							IF aStatCommandQueue[nStatCommandIndex].nSubIndex = 0 THEN
								nStatOffset := 16;
							END_IF;
							nStatElement := 87;
							nStatBitLength := 16;
							bStatSource := False;
							JMP GetInteger;
						END_IF;
						// stProcessDataLimits - nUpper [UINT] [READ_ONLY]
						IF (aStatCommandQueue[nStatCommandIndex].nSubIndex = 0 AND nStatIndex = 1) OR (aStatCommandQueue[nStatCommandIndex].nSubIndex = 2 AND nStatIndex = 0) THEN
							IF aStatCommandQueue[nStatCommandIndex].nSubIndex = 0 THEN
								nStatOffset := 0;
							END_IF;
							nStatElement := 88;
							nStatBitLength := 16;
							bStatSource := False;
							JMP GetInteger;
						END_IF;
				// nSwitchCounter [UINT] [READ_ONLY]
					85:
						nStatComplex := cBASIC_TYPE;
						nStatBitLength := fbReadWriteReq.nCount;
						nStatElement := 89;
						JMP GetInteger;
				// nTemperatureInternal [INT] [READ_ONLY]
					86:
						nStatComplex := cBASIC_TYPE;
						nStatBitLength := fbReadWriteReq.nCount;
						nStatElement := 90;
						JMP GetInteger;
				// stNetwork [ComplexT] [READ_WRITE]
					88:
						nStatComplex := cCOMPLEX_RECORD_TYPE;
						nStatComplexDataTypeSize := UINT_TO_INT(aStatCommandQueue[nStatCommandIndex].nBitLength);
						nStatOffset := 0;
						// stNetwork - nRoleInNetwork [UINT] [READ_WRITE]
						IF (aStatCommandQueue[nStatCommandIndex].nSubIndex = 0 AND nStatIndex = 0) OR (aStatCommandQueue[nStatCommandIndex].nSubIndex = 1 AND nStatIndex = 0) THEN
							IF aStatCommandQueue[nStatCommandIndex].nSubIndex = 0 THEN
								nStatOffset := 8;
							END_IF;
							nStatElement := 91;
							nStatBitLength := 8;
							bStatSource := False;
							JMP GetInteger;
						END_IF;
						// stNetwork - nDeviceNoMasterHighestNo [UINT] [READ_WRITE]
						IF (aStatCommandQueue[nStatCommandIndex].nSubIndex = 0 AND nStatIndex = 1) OR (aStatCommandQueue[nStatCommandIndex].nSubIndex = 2 AND nStatIndex = 0) THEN
							IF aStatCommandQueue[nStatCommandIndex].nSubIndex = 0 THEN
								nStatOffset := 0;
							END_IF;
							nStatElement := 92;
							nStatBitLength := 8;
							bStatSource := False;
							JMP GetInteger;
						END_IF;
			END_CASE;
		END_IF;
		nStatState := cSTATE_JOB_FINISHED;
	END_IF;
// Update FB status
	IF nStatState = cSTATE_JOB_FINISHED THEN
		// Select next command
		nStatCommandIndex := nStatCommandIndex + 1;
		IF (nStatCommandIndex > cNUMBER_INPUTS) OR (aStatCommandQueue[nStatCommandIndex].nIndex = cEMPTY_COMMAND_QUEUE) THEN
			// Job done
			bDone := TRUE;
			bBusy := FALSE;
			bStatBusyMem := FALSE;
			bError := FALSE;
			stErrorCode.nAdsReadError := 16#0000;
			stErrorCode.nAdsWriteError := 16#0000;
			stErrorCode.nIndex := 0;
			stErrorCode.nSubIndex := 0;
			nStatState := cSTATE_READY;
			RETURN;
			// Next command
		ELSE
			nStatState := cSTATE_CLEAR_RECORD; // Send next IO-Link request
		END_IF;
	END_IF;
// End cycle
	RETURN;
// I/O mapping
	// SetInteger
		SetInteger:
			F_Leuze_IOL_SetInteger(nComplex := nStatComplex,
			                 nComplexDataTypeSize := nStatComplexDataTypeSize,
			                 nOffset := nStatOffset,
			                 nSource := nTempDeviceDataInteger,
			                 nBitLength := UINT_TO_INT(nStatBitLength),
			                 aIolRecords := aStatIOLRecords,
			                 aTempItems := aStatTempItems);
			IF (nStatComplex = cBASIC_TYPE) OR (nStatComplex = cCOMPLEX_RECORD_TYPE AND aStatCommandQueue[nStatCommandIndex].nSubIndex > 0) THEN
				fbReadWriteReq(bExecute := TRUE, bRW := TRUE, aData := aStatIOLRecords);
				nStatState := cSTATE_AWAIT_RESPONSE;
			ELSE
				nStatIndex := nStatIndex + 1;
			END_IF;
			RETURN;
	// SetBoolean
		SetBoolean:
			F_Leuze_IOL_SetBoolean(nComplex := nStatComplex,
			                     nComplexDataTypeSize := nStatComplexDataTypeSize,
			                     nOffset := nStatOffset,
			                     bSource := bTempDeviceDataBool,
			                     aIolRecords := aStatIOLRecords,
			                     aTempItems := aStatTempItems);
			IF (nStatComplex = cBASIC_TYPE) OR (nStatComplex = cCOMPLEX_RECORD_TYPE AND aStatCommandQueue[nStatCommandIndex].nSubIndex > 0) THEN
				fbReadWriteReq(bExecute := TRUE, bRW := TRUE, aData := aStatIOLRecords);
				nStatState := cSTATE_AWAIT_RESPONSE;
			ELSE
				nStatIndex := nStatIndex + 1;
			END_IF;
			RETURN;
	// SetString
		SetString:
			F_Leuze_IOL_SetString(nComplex := nStatComplex,
			                   nComplexDataTypeSize := nStatComplexDataTypeSize,
			                   nOffset := nStatOffset,
			                   nfixedLength := UINT_TO_INT(nStatBitLength),
			                   sSource := sTempDeviceDataString,
			                   aIolRecords := aStatIOLRecords,
			                   aTempItems := aStatTempItems);
			IF (nStatComplex = cBASIC_TYPE) OR (nStatComplex = cCOMPLEX_RECORD_TYPE AND aStatCommandQueue[nStatCommandIndex].nSubIndex > 0) THEN
				fbReadWriteReq(bExecute := TRUE, bRW := TRUE, aData := aStatIOLRecords);
				nStatState := cSTATE_AWAIT_RESPONSE;
			ELSE
				nStatIndex := nStatIndex + 1;
			END_IF;
			RETURN;
	// GetInteger
		GetInteger:
			nTempDeviceDataInteger := F_Leuze_IOL_GetInteger(nComplex := nStatComplex,
			                                               nComplexDataTypeSize := nStatComplexDataTypeSize,
			                                               nOffset := nStatOffset,
			                                               nBitLength := UINT_TO_INT(nStatBitLength),
			                                               bIsSigned := bStatSource,
			                                               aIolRecords := aStatIOLRecords,
			                                               aTempItems := aStatTempItems);
			IF nStatComplex = cCOMPLEX_ARRAY_TYPE THEN
				nStatOffset := nStatOffset + 1;
			END_IF;
			CASE nStatElement OF
				23:
						stDeviceData.stData.stDirectParametersPage1.nReserved_1 := DWORD_TO_UINT(nTempDeviceDataInteger);
				24:
						stDeviceData.stData.stDirectParametersPage1.nMasterCycleTime := DWORD_TO_UINT(nTempDeviceDataInteger);
				25:
						stDeviceData.stData.stDirectParametersPage1.nMinCycleTime := DWORD_TO_UINT(nTempDeviceDataInteger);
				26:
						stDeviceData.stData.stDirectParametersPage1.nMSequenceCapability := DWORD_TO_UINT(nTempDeviceDataInteger);
				27:
						stDeviceData.stData.stDirectParametersPage1.nIoLinkRevisionId := DWORD_TO_UINT(nTempDeviceDataInteger);
				28:
						stDeviceData.stData.stDirectParametersPage1.nProcessDataInputLength := DWORD_TO_UINT(nTempDeviceDataInteger);
				29:
						stDeviceData.stData.stDirectParametersPage1.nProcessDataOutputLength := DWORD_TO_UINT(nTempDeviceDataInteger);
				30:
						stDeviceData.stData.stDirectParametersPage1.nVendorId1 := DWORD_TO_UINT(nTempDeviceDataInteger);
				31:
						stDeviceData.stData.stDirectParametersPage1.nVendorId2 := DWORD_TO_UINT(nTempDeviceDataInteger);
				32:
						stDeviceData.stData.stDirectParametersPage1.nDeviceId1 := DWORD_TO_UINT(nTempDeviceDataInteger);
				33:
						stDeviceData.stData.stDirectParametersPage1.nDeviceId2 := DWORD_TO_UINT(nTempDeviceDataInteger);
				34:
						stDeviceData.stData.stDirectParametersPage1.nDeviceId3 := DWORD_TO_UINT(nTempDeviceDataInteger);
				35:
						stDeviceData.stData.stDirectParametersPage1.nReserved_13 := DWORD_TO_UINT(nTempDeviceDataInteger);
				36:
						stDeviceData.stData.stDirectParametersPage1.nReserved_14 := DWORD_TO_UINT(nTempDeviceDataInteger);
				37:
						stDeviceData.stData.stDirectParametersPage1.nReserved_15 := DWORD_TO_UINT(nTempDeviceDataInteger);
				39:
						stDeviceData.stData.stDirectParametersPage2.nDeviceSpecificParameter1 := DWORD_TO_UINT(nTempDeviceDataInteger);
				40:
						stDeviceData.stData.stDirectParametersPage2.nDeviceSpecificParameter2 := DWORD_TO_UINT(nTempDeviceDataInteger);
				41:
						stDeviceData.stData.stDirectParametersPage2.nDeviceSpecificParameter3 := DWORD_TO_UINT(nTempDeviceDataInteger);
				42:
						stDeviceData.stData.stDirectParametersPage2.nDeviceSpecificParameter4 := DWORD_TO_UINT(nTempDeviceDataInteger);
				43:
						stDeviceData.stData.stDirectParametersPage2.nDeviceSpecificParameter5 := DWORD_TO_UINT(nTempDeviceDataInteger);
				44:
						stDeviceData.stData.stDirectParametersPage2.nDeviceSpecificParameter6 := DWORD_TO_UINT(nTempDeviceDataInteger);
				45:
						stDeviceData.stData.stDirectParametersPage2.nDeviceSpecificParameter7 := DWORD_TO_UINT(nTempDeviceDataInteger);
				46:
						stDeviceData.stData.stDirectParametersPage2.nDeviceSpecificParameter8 := DWORD_TO_UINT(nTempDeviceDataInteger);
				47:
						stDeviceData.stData.stDirectParametersPage2.nDeviceSpecificParameter9 := DWORD_TO_UINT(nTempDeviceDataInteger);
				48:
						stDeviceData.stData.stDirectParametersPage2.nDeviceSpecificParameter10 := DWORD_TO_UINT(nTempDeviceDataInteger);
				49:
						stDeviceData.stData.stDirectParametersPage2.nDeviceSpecificParameter11 := DWORD_TO_UINT(nTempDeviceDataInteger);
				50:
						stDeviceData.stData.stDirectParametersPage2.nDeviceSpecificParameter12 := DWORD_TO_UINT(nTempDeviceDataInteger);
				51:
						stDeviceData.stData.stDirectParametersPage2.nDeviceSpecificParameter13 := DWORD_TO_UINT(nTempDeviceDataInteger);
				52:
						stDeviceData.stData.stDirectParametersPage2.nDeviceSpecificParameter14 := DWORD_TO_UINT(nTempDeviceDataInteger);
				53:
						stDeviceData.stData.stDirectParametersPage2.nDeviceSpecificParameter15 := DWORD_TO_UINT(nTempDeviceDataInteger);
				54:
						stDeviceData.stData.stDirectParametersPage2.nDeviceSpecificParameter16 := DWORD_TO_UINT(nTempDeviceDataInteger);
				67:
						stDeviceData.stData.nErrorCount := DWORD_TO_UINT(nTempDeviceDataInteger);
				68:
						stDeviceData.stData.nDeviceStatus := DWORD_TO_UINT(nTempDeviceDataInteger);
				69:
						stDeviceData.stData.stTeachState.nTeachState := DWORD_TO_UINT(nTempDeviceDataInteger);
				70:
						stDeviceData.stData.stSetpoints.nParam1Bdc1Q1 := DWORD_TO_UINT(nTempDeviceDataInteger);
				71:
						stDeviceData.stData.stSetpoints.nParam2Bdc1Q1 := DWORD_TO_UINT(nTempDeviceDataInteger);
				72:
						stDeviceData.stData.stSwitchpointBdc1.nLogic := DWORD_TO_UINT(nTempDeviceDataInteger);
				73:
						stDeviceData.stData.stSwitchpointBdc1.nMode := DWORD_TO_UINT(nTempDeviceDataInteger);
				74:
						stDeviceData.stData.stSwitchpointBdc1.nHysteresis := DWORD_TO_UINT(nTempDeviceDataInteger);
				76:
						stDeviceData.stData.nOnDelaySwitchingOutput := DWORD_TO_UINT(nTempDeviceDataInteger);
				77:
						stDeviceData.stData.nOffDelaySwitchingOutput := DWORD_TO_UINT(nTempDeviceDataInteger);
				78:
						stDeviceData.stData.nMultiIOPin4 := DWORD_TO_UINT(nTempDeviceDataInteger);
				79:
						stDeviceData.stData.nMultiIOPin2 := DWORD_TO_UINT(nTempDeviceDataInteger);
				80:
						stDeviceData.stData.stAnalogRange.nLowerLimit := DWORD_TO_UINT(nTempDeviceDataInteger);
				81:
						stDeviceData.stData.stAnalogRange.nUpperLimit := DWORD_TO_UINT(nTempDeviceDataInteger);
				82:
						stDeviceData.stData.nTemperatureCompensation := DWORD_TO_UINT(nTempDeviceDataInteger);
				83:
						stDeviceData.stData.stTeachpointSp1.nTp1 := DWORD_TO_UINT(nTempDeviceDataInteger);
				84:
						stDeviceData.stData.stTeachpointSp1.nTp2 := DWORD_TO_UINT(nTempDeviceDataInteger);
				85:
						stDeviceData.stData.stTeachpointSp2.nTp1 := DWORD_TO_UINT(nTempDeviceDataInteger);
				86:
						stDeviceData.stData.stTeachpointSp2.nTp2 := DWORD_TO_UINT(nTempDeviceDataInteger);
				87:
						stDeviceData.stData.stProcessDataLimits.nLower := DWORD_TO_UINT(nTempDeviceDataInteger);
				88:
						stDeviceData.stData.stProcessDataLimits.nUpper := DWORD_TO_UINT(nTempDeviceDataInteger);
				89:
						stDeviceData.stData.nSwitchCounter := DWORD_TO_UINT(nTempDeviceDataInteger);
				90:
						stDeviceData.stData.nTemperatureInternal := DWORD_TO_INT(nTempDeviceDataInteger);
				91:
						stDeviceData.stData.stNetwork.nRoleInNetwork := DWORD_TO_UINT(nTempDeviceDataInteger);
				92:
						stDeviceData.stData.stNetwork.nDeviceNoMasterHighestNo := DWORD_TO_UINT(nTempDeviceDataInteger);
			END_CASE;
			IF (nStatComplex = cBASIC_TYPE) OR (nStatComplex = cCOMPLEX_RECORD_TYPE AND aStatCommandQueue[nStatCommandIndex].nSubIndex > 0) THEN
				nStatState := cSTATE_JOB_FINISHED;
			ELSE
				nStatIndex := nStatIndex + 1;
			END_IF;
			RETURN;
	// GetString
		GetString:
			sTempDeviceDataString := F_Leuze_IOL_GetString(nComplex := nStatComplex,
			                                        nComplexDataTypeSize := nStatComplexDataTypeSize,
			                                        nOffset := nStatOffset,
			                                        nfixedLength := UINT_TO_INT(nStatBitLength),
			                                        aIolRecords := aStatIOLRecords,
			                                        aTempItems := aStatTempItems);
			IF nStatComplex = cCOMPLEX_ARRAY_TYPE THEN
				nStatOffset := nStatOffset + 1;
			END_IF;
			CASE nStatElement OF
				60:
						stDeviceData.stData.sVendorName := sTempDeviceDataString;
				61:
						stDeviceData.stData.sVendorText := sTempDeviceDataString;
				62:
						stDeviceData.stData.sProductName := sTempDeviceDataString;
				63:
						stDeviceData.stData.sProductId := sTempDeviceDataString;
				64:
						stDeviceData.stData.sProductText := sTempDeviceDataString;
				65:
						stDeviceData.stData.sFirmwareRevision := sTempDeviceDataString;
				66:
						stDeviceData.stData.sApplicationSpecificTag := sTempDeviceDataString;
				75:
						stDeviceData.stData.sLot := sTempDeviceDataString;
			END_CASE;
			IF nStatComplex = cBASIC_TYPE THEN
				nStatState := cSTATE_JOB_FINISHED;
			ELSE
				nStatIndex := nStatIndex + 1;
			END_IF;
			RETURN;
	// GetBoolean
		GetBoolean:
			bTempDeviceDataBool := F_Leuze_IOL_GetBoolean(nComplex := nStatComplex,
			                                       nComplexDataTypeSize := nStatComplexDataTypeSize,
			                                       nOffset := nStatOffset,
			                                       aIolRecords := aStatIOLRecords,
			                                       aTempItems := aStatTempItems);
			IF nStatComplex = cCOMPLEX_ARRAY_TYPE THEN
				nStatOffset := nStatOffset + 1;
			END_IF;
			CASE nStatElement OF
				56:
						stDeviceData.stData.stDeviceAccessLocks.bParameterWriteAccess := bTempDeviceDataBool;
				57:
						stDeviceData.stData.stDeviceAccessLocks.bDataStorage := bTempDeviceDataBool;
				58:
						stDeviceData.stData.stDeviceAccessLocks.bLocalParameterization := bTempDeviceDataBool;
				59:
						stDeviceData.stData.stDeviceAccessLocks.bLocalUserInterface := bTempDeviceDataBool;
			END_CASE;
			IF (nStatComplex = cBASIC_TYPE) OR (nStatComplex = cCOMPLEX_RECORD_TYPE AND aStatCommandQueue[nStatCommandIndex].nSubIndex > 0) THEN
				nStatState := cSTATE_JOB_FINISHED;
			ELSE
				nStatIndex := nStatIndex + 1;
			END_IF;
			RETURN;

END_FUNCTION_BLOCK
